FUNCTION_BLOCK CPress_HMI (* Service Interface Function Block Type *)
  (* Standard: 61499-2 *)
  (* Version 0.0, 30/03/2026, template *)
  PACKAGE Hidryco.HidrycoLib;
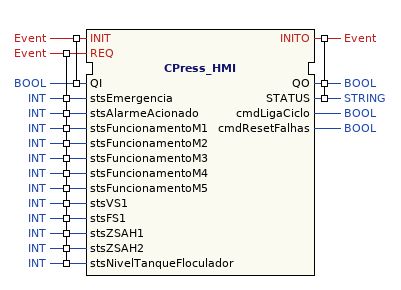
  EVENT_INPUT
    INIT WITH QI;
    REQ WITH stsEmergencia, stsAlarmeAcionado, stsFuncionamentoM1, stsFuncionamentoM2, stsFuncionamentoM3, stsFuncionamentoM4, stsFuncionamentoM5, stsVS1, stsFS1, stsZSAH1, stsZSAH2, stsNivelTanqueFloculador;
  END_EVENT
  EVENT_OUTPUT
    INITO WITH QO, STATUS;
  END_EVENT
  VAR_INPUT
    QI : BOOL;
    stsEmergencia : INT;
    stsAlarmeAcionado : INT; (* Alarme H *)
    stsFuncionamentoM1 : INT; (* Funcionamento da prensa M1. *)
    stsFuncionamentoM2 : INT; (* Funcionamento do moto redutor limpeza M2 *)
    stsFuncionamentoM3 : INT; (* Funcionamento do agitador floculador M3 *)
    stsFuncionamentoM4 : INT; (* Funcionamento da bomba de água M4 *)
    stsFuncionamentoM5 : INT; (* Funcionamento do compressor M5 *)
    stsVS1 : INT; (* Status da válvula solenoide de limpeza VS1 *)
    stsFS1 : INT; (* Status chave de fluxo FS1 *)
    stsZSAH1 : INT; (* Fim de curso frontal limpeza ZSAH1 *)
    stsZSAH2 : INT; (* Fim de curso trazeira limpeza ZSAH2 *)
    stsNivelTanqueFloculador : INT;
  END_VAR
  VAR_OUTPUT
    QO : BOOL; (* Event Output Qualifier *)
    STATUS : STRING; (* Service Status *)
    cmdLigaCiclo : BOOL;
    cmdResetFalhas : BOOL;
  END_VAR
  SERVICE /
    SEQUENCE 
    END_SEQUENCE
  END_SERVICE
END_FUNCTION_BLOCK
